TYPE PAL_Busy :
(
	ePALStart := 0
	
	
);
END_TYPE

(* stored: Version 1.1.0.1, ProductVersion 3.1.4024.2
   DUT PAL_Busy: Id {175432ff-b200-404b-8a01-65439cb39b54} *)
